FUNCTION_BLOCK OUT_ANY_CONSOLE (* Service Interface Function Block Type for debugging, tracing, etc. *)
  (* Compiler Cpp Unknown Unknown 1.0 *)
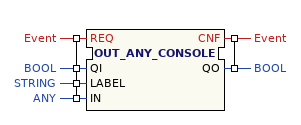
  EVENT_INPUT
    REQ WITH QI, IN, LABEL; (* Service Request *)
  END_EVENT
  EVENT_OUTPUT
    CNF WITH QO; (* Confirmation of Requested Service *)
  END_EVENT
  VAR_INPUT
    QI : BOOL; (* Event Input Qualifier *)
    LABEL : STRING; (* Label for the output value *)
    IN : ANY; (* Output value to console *)
  END_VAR
  VAR_OUTPUT
    QO : BOOL; (* Event Output Qualifier *)
  END_VAR
END_FUNCTION_BLOCK
